// TIA Portal V20 export
TYPE "typeCmControlNodeSoftCam"
// stored: Namespace Unit1.Em2
   STRUCT
      jrOutPnPLeftAxisX : "Unit1.Em2.typeCmControlNodeSoftCamjrOutPnPLeftAxisX";
      jrOutPnPLeftAxisZ : "Unit1.Em2.typeCmControlNodeSoftCamjrOutPnPLeftAxisZ";
      jrOutPnPRightAxisX : "Unit1.Em2.typeCmControlNodeSoftCamjrOutPnPRightAxisX";
      jrOutPnPRightAxisZ : "Unit1.Em2.typeCmControlNodeSoftCamjrOutPnPRightAxisZ";
   END_STRUCT;
END_TYPE
